{attribute 'GeneratedUsingTerminal: EK1100-0000-0018'}
{attribute addProperty BoxType "EK1100-0000-0018"}
{attribute addProperty Id "Beckhoff_EPP3xxxEK1122Beckhoff_EPP3xxxEK1122_998B9B3E1480"}
{attribute addProperty CRC "1073152268"}
{attribute addProperty Size "1480"}
TYPE Beckhoff_EPP3xxx_3FF7010C EXTENDS EK1100_1FC0878B :
STRUCT
	{attribute addProperty Name "Beckhoff_EPP3xxxEK1122"}
	{attribute addProperty PreviousPort "Beckhoff EPP3xxx : B"}
	Beckhoff_EPP3xxxEK1122 : Beckhoff_EPP3xxxEK1122_998B9B3E;
END_STRUCT
END_TYPE

(* stored: Version 1.2.0.0, ProductVersion 3.1.4024.9
   DUT Beckhoff_EPP3xxx_3FF7010C: Id {b88ad8d5-9ebc-49e4-afdf-492a6e6a46ad} *)
